{attribute 'qualified_only'}
{attribute 'strict'}
{attribute 'to_string'}
TYPE E_Modes :
(	
	Manuel := 1,
	Off := 2,
	Auto := 3
);
END_TYPE

(* stored: Version 1.1.0.1
   DUT E_Modes: Id {e868f847-14a4-46b6-9a53-b54aff0f5a8f} *)
